// TIA Portal V17 export
ORGANIZATION_BLOCK "Main"   // OB1, LAD
BEGIN
END_ORGANIZATION_BLOCK
